FUNCTION_BLOCK Revezamento_3_Motores_HMI (* Service Interface Function Block Type *)
  (* Standard: 61499-2 *)
  (* Version 0.0, 25/02/2026, template *)
  PACKAGE Hidryco.HidrycoLib;
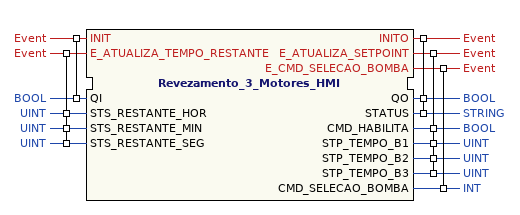
  EVENT_INPUT
    INIT WITH QI;
    E_ATUALIZA_TEMPO_RESTANTE WITH STS_RESTANTE_HOR, STS_RESTANTE_MIN, STS_RESTANTE_SEG;
  END_EVENT
  EVENT_OUTPUT
    INITO WITH QO, STATUS;
    E_ATUALIZA_SETPOINT WITH CMD_HABILITA, STP_TEMPO_B1, STP_TEMPO_B2, STP_TEMPO_B3;
    E_CMD_SELECAO_BOMBA WITH CMD_SELECAO_BOMBA;
  END_EVENT
  VAR_INPUT
    QI : BOOL;
    STS_RESTANTE_HOR : UINT;
    STS_RESTANTE_MIN : UINT;
    STS_RESTANTE_SEG : UINT;
  END_VAR
  VAR_OUTPUT
    QO : BOOL; (* Event Output Qualifier *)
    STATUS : STRING; (* Service Status *)
    CMD_HABILITA : BOOL;
    STP_TEMPO_B1 : UINT;
    STP_TEMPO_B2 : UINT;
    STP_TEMPO_B3 : UINT;
    CMD_SELECAO_BOMBA : INT;
  END_VAR
  SERVICE /
    SEQUENCE 
    END_SEQUENCE
  END_SERVICE
END_FUNCTION_BLOCK
